Staubli VAL3: STRALIGN.pgx

public program strAlign(string& x_sStrIn[], num x_nLength, string x_sAlign, string x_sChar)
  local num l_i
  local num l_nToAdd
  local num l_nAscii
begin
  // This program modify the input string to align it
  // left,right or centered
  //
  // Input Param
  // x_sStrIn   : Input string to modify
  // x_nLength  : Length of the output string
  // x_sAlign   : Align mode
  //                  : C-c = Centered
  //                    L-l = Align Left
  //                    R-r = Align Right
  switch x_sAlign
    // Centered
    case "C","c"
      if len(x_sStrIn)<x_nLength
        l_nToAdd=x_nLength-len(x_sStrIn)
      endIf
    break
    // Left
    case "L","l"
      if len(x_sStrIn)<x_nLength
        l_nToAdd=x_nLength-len(x_sStrIn)
        for l_i=1 to l_nToAdd
          x_sStrIn=x_sStrIn+x_sChar
        endFor
      else
        x_sStrIn=mid(x_sStrIn,x_nLength,0)
      endIf
    break
    // Right
    case "R","r"
      if len(x_sStrIn)<x_nLength
        l_nToAdd=x_nLength-len(x_sStrIn)
        for l_i=1 to l_nToAdd
          x_sStrIn=x_sChar+x_sStrIn
        endFor
      else
        x_sStrIn=mid(x_sStrIn,x_nLength,0)
      endIf
    break
  endSwitch
end
